FUNCTION_BLOCK FB_HeightMeasurement2
VAR_INPUT
	
	aSensorCurrentValue							: ARRAY[1..4] OF REAL;		
	bEnable										: BOOL;
	bMeasurementRequest							: BOOL;
	bManualMode									: BOOL;
	bSetFixedPoints								: BOOL;
	aTolerance									: ARRAY[1..3] OF REAL;
	
	bAcknowledge								: BOOL;
	
	//Calibration block
	
	nDistanceBetweenPoints						: ARRAY[1..3] OF REAL;
	anDistanceSetPoint							: ARRAY[1..3] OF REAL;
	
	
	
	
					
END_VAR
VAR_OUTPUT
	
	bBusy										: BOOL;
	bComplete									: BOOL;
	bEnableo									: BOOL;
	aPass										: ARRAY[1..5] OF BOOL; //5 Final Result
	aFail										: ARRAY[1..5] OF BOOL; //5 Final Result
	aMinLimitCalibrationBlock					: ARRAY[1..3] OF REAL;
	aMaxLimitCalibrationBlock					: ARRAY[1..3] OF REAL;
	
	aDistanceBetweenProbes						: ARRAY[1..3] OF REAL; //1 Probe 1 to probe zero
	abSensorStuck								: ARRAY[1..4] OF BOOL;
	nFixedPoint									: ARRAY[1..4] OF REAL;
	aScaledSensorCurrentValue					: ARRAY[1..4] OF REAL;
	
	nHeightMeasureStateValue					: ARRAY[1..4] OF DINT;

	

END_VAR
VAR PERSISTENT
	
	nSensorSetPoint								: ARRAY[1..4] OF REAL;
	
END_VAR
VAR
	
	i											: INT;
	j											: INT;
	tonTestingTime								: TON;
	rMeasurementRequest							: R_TRIG;
	nHeightOffset								: REAL;
	
	EHeighttMeasureProcess						: E_HeighttMeasureProcess;
	anValueBeforeMeasurement					: ARRAY[1..4] OF REAL;
	
	
END_VAR

ACT_ScaleMinMax();
ACT_SetPoints();

IF NOT bEnable THEN
	EHeighttMeasureProcess						:= E_HeighttMeasureProcess.WAITING_ENABLE;
ELSIF bManualMode AND bEnable THEN
	EHeighttMeasureProcess						:= E_HeighttMeasureProcess.Manual_Mode;
END_IF
bEnableo										:= bEnable;
tonTestingTime( IN := (EHeighttMeasureProcess = E_HeighttMeasureProcess.WAITING_FOR_MEASURE), PT := T#3S);
rMeasurementRequest( CLK := bMeasurementRequest);

CASE EHeighttMeasureProcess OF

E_HeighttMeasureProcess.WAITING_ENABLE:

	IF bEnable THEN
		EHeighttMeasureProcess					:= E_HeighttMeasureProcess.WAITING_MEASURING_REQUEST;
	END_IF

E_HeighttMeasureProcess.WAITING_MEASURING_REQUEST:	

	bComplete									:= FALSE;
	IF rMeasurementRequest.Q THEN
		EHeighttMeasureProcess					:= E_HeighttMeasureProcess.RESET;
	END_IF
	
	anValueBeforeMeasurement					:= aSensorCurrentValue;

E_HeighttMeasureProcess.RESET:
	
	
	abSensorStuck[1]							:= FALSE;
	
	FOR i := 1 TO 5 DO
		aPass[i]								:= FALSE;	
		aFail[i]								:= FALSE;
	END_FOR
	FOR j := 1 TO 3 DO
		nHeightMeasureStateValue[j]				:= 0;
	END_FOR
		EHeighttMeasureProcess					:= E_HeighttMeasureProcess.WAITING_FOR_MEASURE;
	
E_HeighttMeasureProcess.SENSOR_STUCK_EVALUATION:

	ACT_SensorStuck();
	
E_HeighttMeasureProcess.WAITING_FOR_MEASURE:

	IF tonTestingTime.Q  THEN
		EHeighttMeasureProcess					:= E_HeighttMeasureProcess.CALIBRATIONBLOCK_METHOD;
	END_IF

E_HeighttMeasureProcess.CALIBRATIONBLOCK_METHOD:

		ACT_CalibrationBlockMethod();
		bComplete								:= TRUE;
		IF bAcknowledge THEN
			EHeighttMeasureProcess					:= E_HeighttMeasureProcess.WAITING_MEASURING_REQUEST;
		END_IF

E_HeighttMeasureProcess.Manual_Mode:
		
		ACT_ManualMode();		

END_CASE


bBusy				:= 	(EHeighttMeasureProcess	<> E_HeighttMeasureProcess.WAITING_ENABLE AND
						EHeighttMeasureProcess  <> E_HeighttMeasureProcess.WAITING_MEASURING_REQUEST) AND
						NOT bComplete;

ACTION ACT_CalibrationBlockMethod:
aDistanceBetweenProbes[1] 	:= (nFixedPoint[4] - aScaledSensorCurrentValue[4])+ (aScaledSensorCurrentValue[1] - (nFixedPoint[1])) + nDistanceBetweenPoints[1];
aDistanceBetweenProbes[2] 	:= (nFixedPoint[4] - aScaledSensorCurrentValue[4])+ (aScaledSensorCurrentValue[2] - (nFixedPoint[2])) + nDistanceBetweenPoints[2];
aDistanceBetweenProbes[3] 	:= (nFixedPoint[4] - aScaledSensorCurrentValue[4])+ (aScaledSensorCurrentValue[3] - (nFixedPoint[3])) + nDistanceBetweenPoints[3];

FOR i := 1 TO 3 DO
	IF (aDistanceBetweenProbes[i] <= aMaxLimitCalibrationBlock[i]) AND (aDistanceBetweenProbes[i] >= aMinLimitCalibrationBlock[i]) THEN
		
		aPass[i]			:= TRUE;
		nHeightMeasureStateValue[i] := 1;
	ELSE 
		aFail[i]			:= TRUE;
		nHeightMeasureStateValue[i] := 2;
	END_IF
END_FOR

IF aPass[1] AND aPass[2] AND aPass[3] THEN
	aPass[5]			:= TRUE;
ELSIF aFail[1] OR aFail[2] OR aFail[3] THEN
	aFail[5]			:= TRUE;
END_IF
END_ACTION

ACTION ACT_ManualMode:
aDistanceBetweenProbes[1] 	:= (nFixedPoint[4] - aScaledSensorCurrentValue[4])+ (aScaledSensorCurrentValue[1] - (nFixedPoint[1])) + nDistanceBetweenPoints[1];
aDistanceBetweenProbes[2] 	:= (nFixedPoint[4] - aScaledSensorCurrentValue[4])+ (aScaledSensorCurrentValue[2] - (nFixedPoint[2])) + nDistanceBetweenPoints[2];
aDistanceBetweenProbes[3] 	:= (nFixedPoint[4] - aScaledSensorCurrentValue[4])+ (aScaledSensorCurrentValue[3] - (nFixedPoint[3])) + nDistanceBetweenPoints[3];

IF (aDistanceBetweenProbes[1] <= aMaxLimitCalibrationBlock[1]) AND (aDistanceBetweenProbes[1] >= aMinLimitCalibrationBlock[1]) THEN
	
		nHeightMeasureStateValue[1] := 1;
ELSE 
		nHeightMeasureStateValue[1] := 2;
END_IF

IF (aDistanceBetweenProbes[2] <= aMaxLimitCalibrationBlock[2]) AND (aDistanceBetweenProbes[2] >= aMinLimitCalibrationBlock[2]) THEN
	
		nHeightMeasureStateValue[2] := 1;
ELSE 
		nHeightMeasureStateValue[2] := 2;
END_IF

IF (aDistanceBetweenProbes[3] <= aMaxLimitCalibrationBlock[3]) AND (aDistanceBetweenProbes[3] >= aMinLimitCalibrationBlock[3]) THEN
	
		nHeightMeasureStateValue[3] := 1;
ELSE 
		nHeightMeasureStateValue[3] := 2;
END_IF
END_ACTION

ACTION ACT_ScaleMinMax:
//Current value SCALE
IF aSensorCurrentValue[1] <> 0 THEN
	
	aScaledSensorCurrentValue[1]		:= aSensorCurrentValue[1]/10000;
	
ELSE aScaledSensorCurrentValue[1]		:= 0;

END_IF

IF aSensorCurrentValue[2] <> 0 THEN
	
	aScaledSensorCurrentValue[2]		:= aSensorCurrentValue[2]/10000;
	
ELSE aScaledSensorCurrentValue[2]		:= 0;

END_IF

IF aSensorCurrentValue[3] <> 0 THEN
	
	aScaledSensorCurrentValue[3]		:= aSensorCurrentValue[3]/10000;
	
ELSE aScaledSensorCurrentValue[3]		:= 0;

END_IF

IF aSensorCurrentValue[4] <> 0 THEN
	
	aScaledSensorCurrentValue[4]		:= aSensorCurrentValue[4]/10000;
	
ELSE aScaledSensorCurrentValue[4]		:= 0;

END_IF

aMaxLimitCalibrationBlock[1]			:= anDistanceSetPoint[1] + aTolerance[1];
aMaxLimitCalibrationBlock[2]			:= anDistanceSetPoint[2] + aTolerance[2];
aMaxLimitCalibrationBlock[3]			:= anDistanceSetPoint[3] + aTolerance[3];

aMinLimitCalibrationBlock[1]			:= anDistanceSetPoint[1] - aTolerance[1];
aMinLimitCalibrationBlock[2]			:= anDistanceSetPoint[2] - aTolerance[2];
aMinLimitCalibrationBlock[3]			:= anDistanceSetPoint[3] - aTolerance[3];
END_ACTION

ACTION ACT_SensorStuck:
IF (anValueBeforeMeasurement[1] <= (aSensorCurrentValue[1] + 0.5)) AND (anValueBeforeMeasurement[1] >= (aSensorCurrentValue[1] - 0.5)) THEN
		abSensorStuck[1]							:= TRUE;
	END_IF

IF (anValueBeforeMeasurement[2] <= (aSensorCurrentValue[2] + 0.5)) AND (anValueBeforeMeasurement[2] >= (aSensorCurrentValue[2] - 0.5)) THEN
		abSensorStuck[2]							:= TRUE;
	END_IF

IF (anValueBeforeMeasurement[3] <= (aSensorCurrentValue[3] + 0.5)) AND (anValueBeforeMeasurement[3] >= (aSensorCurrentValue[3] - 0.5)) THEN
		abSensorStuck[3]							:= TRUE;
	END_IF

IF (anValueBeforeMeasurement[4] <= (aSensorCurrentValue[4] + 0.5)) AND (anValueBeforeMeasurement[4] >= (aSensorCurrentValue[4] - 0.5)) THEN
		abSensorStuck[4]							:= TRUE;
	END_IF
END_ACTION

ACTION ACT_SetPoints:
IF bSetFixedPoints THEN
	
	nSensorSetPoint[1]						:= aScaledSensorCurrentValue[1];
	nSensorSetPoint[2]						:= aScaledSensorCurrentValue[2];
	nSensorSetPoint[3]						:= aScaledSensorCurrentValue[3];
	nSensorSetPoint[4]						:= aScaledSensorCurrentValue[4];
ELSE
	
	nFixedPoint[1]							:= nSensorSetPoint[1];
	nFixedPoint[2]							:= nSensorSetPoint[2];
	nFixedPoint[3]							:= nSensorSetPoint[3];
	nFixedPoint[4]							:= nSensorSetPoint[4];



END_IF
END_ACTION

END_FUNCTION_BLOCK

(* stored: Version 1.1.0.1, ProductVersion 3.1.4024.13
   POU FB_HeightMeasurement2: Id {46e18333-d1f7-4aac-b31b-53a6366d4c44}, SpecialFunc None
   Action ACT_CalibrationBlockMethod: Id {b9a3cda6-aa2b-4bef-a9fd-5776bf0537cb}
   Action ACT_ManualMode: Id {4dc37cac-4f9f-4d57-97db-a1bcf016dafb}
   Action ACT_ScaleMinMax: Id {c6383b02-bb9e-45e4-85ac-68840cd6851a}
   Action ACT_SensorStuck: Id {97d66adc-213d-4544-88ac-fa4ee0417671}
   Action ACT_SetPoints: Id {f1eba2c3-d13a-4104-821d-56df975234b4} *)
